Yaskawa INFORM job: KRIS8-PODLUZNCA_NEW.JBI

/JOB
//NAME KRIS8-PODLUZNCA_NEW
//POS
///NPOS 200,200,200,13,0,0
///TOOL 0
///POSTYPE PULSE
///PULSE
C00000=1998,-113620,-91819,0,89171,2
C00001=1998,-113620,-91819,0,89171,2
C00002=1998,-113620,-91819,0,89171,2
C00003=-50148,47658,9015,-3478,103612,-52965
C00004=-87671,10112,-26644,4452,101827,-68771
C00005=-89510,7784,-25446,4619,99998,-69437
C00006=-89510,7526,-24742,4610,99434,-69459
C00007=-89510,7784,-25446,4619,99998,-69437
C00008=-89141,5759,-27209,4581,100025,-69316
C00009=-89510,7784,-25446,4619,99998,-69437
C00010=-118549,-7920,-36001,7391,100506,-78970
C00011=-118558,-8065,-31852,7324,97901,-79128
C00012=-118558,-8215,-30981,7313,97294,-79164
C00013=-118558,-8065,-31852,7324,97901,-79128
C00014=-118526,-10509,-33773,7321,97825,-79123
C00015=-118558,-8065,-31852,7324,97901,-79128
C00016=-118558,-6729,-36855,7427,101637,-78904
C00017=-99982,-14384,-32914,3812,87667,-73559
C00018=-100648,-9156,-23354,4670,87204,-73724
C00019=-100648,-9135,-22594,4670,86748,-73740
C00020=-100648,-9156,-23354,4670,87204,-73724
C00021=-100304,-11982,-25556,4620,87088,-73613
C00022=-100648,-9156,-23354,4670,87204,-73724
C00023=-126523,-14506,-29918,8084,90525,-82231
C00024=-126543,-14617,-21806,8089,85527,-82559
C00025=-126543,-14515,-21015,8091,85096,-82587
C00026=-126543,-14617,-21806,8089,85527,-82559
C00027=-126622,-16805,-23452,8098,85423,-82593
C00028=-126543,-14617,-21806,8089,85527,-82559
C00029=-126543,-15095,-29845,8084,90184,-82258
C00030=-141008,-142584,-88347,10734,62671,-89412
C00031=-2633,-142584,-88347,10734,62671,-89412
C00032=-538,152103,58256,11565,122730,-83592
C00033=-538,152103,58256,11565,122730,-83592
C00034=-538,163731,66428,11721,123660,-83483
C00035=-24110,80646,-6840,3666,118579,-81953
C00036=-70155,49076,-66751,3666,118579,-81953
C00037=-75302,69312,-21887,-16743,132273,-74648
C00038=-73641,66162,-19190,-16029,129345,-73576
C00039=-73641,65328,-19214,-15924,128944,-73508
C00040=-74175,68002,-17054,-15046,130211,-73509
C00041=-73715,66523,-18896,-15177,130633,-73426
C00042=-74175,68002,-17054,-15046,130211,-73509
C00043=-74175,75772,-16365,-16008,133654,-74118
C00044=-92792,60028,-40452,-15957,137944,-80854
C00045=-92792,54549,-41170,-15193,135653,-80408
C00046=-92792,53504,-41275,-15052,135198,-80323
C00047=-92792,54549,-41170,-15193,135653,-80408
C00048=-92488,53114,-42914,-15337,136011,-80380
C00049=-92792,54549,-41170,-15193,135653,-80408
C00050=-92792,27665,-39260,-12049,121058,-78294
C00051=-132608,13603,-46395,-6888,114515,-90217
C00052=-132421,12280,-41624,-6966,112053,-90060
C00053=-132421,11796,-41286,-6941,111598,-90034
C00054=-132421,12280,-41624,-6966,112053,-90060
C00055=-132588,9844,-43810,-6954,112133,-90118
C00056=-132421,12280,-41624,-6966,112053,-90060
C00057=-132421,20626,-45689,-7423,118793,-90495
C00058=-93642,14896,-51087,-11726,122768,-78621
C00059=-121167,7250,-60994,-9109,122189,-87287
C00060=-121133,19973,-49305,-9042,121542,-87220
C00061=-121132,14285,-46771,-8609,117111,-86854
C00062=-121132,13713,-46508,-8571,116661,-86819
C00063=-121132,14285,-46771,-8609,117111,-86854
C00064=-121135,12460,-48440,-8614,117198,-86860
C00065=-121132,14285,-46771,-8609,117111,-86854
C00066=-121132,17545,-48059,-8835,119552,-87051
C00067=-132875,22669,-43773,5943,121981,-86806
C00068=-135068,19005,-43202,8732,120135,-86865
C00069=-125533,16786,-42812,7853,119266,-83887
C00070=-129035,15453,-41030,19832,117551,-82149
C00071=-130355,18004,-41916,20330,119568,-82220
C00072=-130907,11274,-51649,20974,122055,-81903
C00073=-97666,14619,-44772,-31513,122541,-85138
C00074=-89089,20309,-29812,-48880,120265,-85971
C00075=-90138,26219,-24118,-48560,119457,-86029
C00076=-94354,21466,-28820,-38570,118301,-84723
C00077=-94339,20725,-28307,-38311,117755,-84491
C00078=-97943,20254,-33169,-26633,118711,-83166
C00079=-102801,18851,-37203,-11200,118340,-81013
C00080=-105344,17460,-38317,-1076,116820,-79338
C00081=-107629,15720,-38660,7756,114602,-78025
C00082=-107337,17368,-35211,13069,113626,-76697
C00083=-107325,21456,-38051,13546,117374,-76240
C00084=-114827,9197,-39078,13016,110805,-79564
C00085=-114816,5999,-36185,12673,107231,-79960
C00086=-89500,15411,-20924,8846,98241,-72558
C00087=-89521,17497,-24405,8955,101422,-72333
C00088=-120014,-138037,-117853,25062,55116,-87984
C00089=-139340,-34559,-66869,29462,80713,-89295
C00090=-144770,-30804,-73292,39943,77473,-90359
C00091=-143362,-21275,-66712,39157,77581,-89780
C00092=-144483,-24614,-74965,39351,80645,-89055
C00093=-151238,-55243,-102038,42556,83965,-90229
C00094=10330,-8063,-71326,-50992,95178,-51096
C00095=10330,-154777,-122755,75707,95178,-51096
C00096=10330,-154777,-122755,75707,95178,-51096
C00097=-84612,8206,-36800,5840,103129,-68484
C00098=-86865,7918,-29603,3944,101662,-68585
C00099=-87828,11476,-22006,5366,101518,-68689
C00100=-118917,-5972,-29345,7466,99945,-79124
C00101=-118924,-4449,-32352,7580,103027,-78936
C00102=-137167,-2659,-36348,8728,105802,-84843
C00103=-109963,-5720,-34048,6846,100758,-76100
C00104=-138502,-3992,-26225,8429,99500,-85759
C00105=-138502,843,-39441,8925,110003,-85001
C00106=-88254,-47088,-61974,-10192,62970,-70123
C00107=-81608,-29587,-43634,-21841,66061,-69208
C00108=-83532,-22198,-38463,-20877,66146,-69964
C00109=-81853,-28331,-46732,-21354,68381,-69747
C00110=-4657,-138190,-117116,-41247,88176,-44256
C00111=1998,-113620,-91819,0,89171,2
C00112=-50148,47658,9015,-3478,103612,-52965
C00113=-122206,-8197,-37642,7697,101693,-80109
C00114=-122172,-5530,-28898,7592,99531,-80240
C00115=-122172,-5644,-28166,7579,99029,-80270
C00116=-122172,-5530,-28898,7592,99531,-80240
C00117=-122187,-7349,-30356,7592,99495,-80247
C00118=-122172,-5530,-28898,7592,99531,-80240
C00119=-152388,7436,-14473,8976,99151,-90470
C00120=-152540,6439,-11770,9191,96395,-90696
C00121=-152540,6437,-10968,9184,95908,-90732
C00122=-152540,6439,-11770,9191,96395,-90696
C00123=-152857,4706,-13266,9200,96461,-90799
C00124=-152540,6439,-11770,9191,96395,-90696
C00125=-152540,6878,-17750,9308,100253,-90406
C00126=-127365,-8235,-30314,7954,97587,-82094
C00127=-127365,-8135,-15746,8070,86282,-82798
C00128=-127365,-8012,-14852,8071,85798,-82829
C00129=-127365,-8135,-15746,8070,86282,-82798
C00130=-127450,-10284,-17434,8077,86227,-82833
C00131=-127365,-8135,-15746,8070,86282,-82798
C00132=-126523,-14506,-29918,8084,90525,-82231
C00133=-123077,-8463,-14980,-23626,83972,-82532
C00134=-125016,-5406,-1705,-27943,77200,-81831
C00135=-125016,-5123,-715,-27989,76788,-81729
C00136=-125016,-5449,-1860,-27937,77265,-81847
C00137=-125063,-7239,-3294,-27936,77216,-81852
C00138=-125016,-5449,-1860,-27937,77265,-81847
C00139=-125016,-6433,-5581,-27781,78853,-82232
C00140=-141008,-142584,-88347,10734,62671,-89412
C00141=-2633,-142584,-88347,10734,62671,-89412
C00142=-538,152103,58256,11565,122730,-83592
C00143=-538,152103,58256,11565,122730,-83592
C00144=-538,163731,66428,11721,123660,-83483
C00145=-24110,80646,-6840,3666,118579,-81953
C00146=-70155,49076,-66751,3666,118579,-81953
C00147=-75302,69312,-21887,-16743,132273,-74648
C00148=-71157,73317,-9100,-15659,127243,-72407
C00149=-71157,72393,-9111,-15553,126791,-72333
C00150=-71157,73317,-9100,-15659,127243,-72407
C00151=-70763,72072,-10673,-15771,127615,-72338
C00152=-71157,73317,-9100,-15659,127243,-72407
C00153=-71157,75512,-9016,-15913,128280,-72581
C00154=-70753,69276,-8084,9618,109691,-64304
C00155=-70054,68719,-6250,9333,108233,-64227
C00156=-70054,67798,-6136,9301,107694,-64269
C00157=-70054,68719,-6250,9333,108233,-64227
C00158=-69682,67506,-7733,9249,108486,-64104
C00159=-70054,68719,-6250,9333,108233,-64227
C00160=-71410,68261,-9608,9830,110161,-64447
C00161=-100211,16967,-41384,-5250,115146,-78637
C00162=-100101,13848,-40894,-5174,113254,-78516
C00163=-100101,13093,-40376,-5142,112548,-78482
C00164=-100101,13848,-40894,-5174,113254,-78516
C00165=-99916,12326,-42277,-5198,113335,-78462
C00166=-100101,13848,-40894,-5174,113254,-78516
C00167=-128373,12968,-45365,-6146,114904,-88569
C00168=-128373,11236,-44374,-6065,113413,-88488
C00169=-128373,10392,-43832,-6025,112650,-88447
C00170=-128373,11236,-44374,-6065,113413,-88488
C00171=-128461,9274,-46126,-6059,113476,-88521
C00172=-128373,11236,-44374,-6065,113413,-88488
C00173=-126467,9541,-45537,-4537,113892,-87464
C00174=-90696,17389,-28668,-7563,109954,-75731
C00175=-90696,19081,-30431,-7676,111892,-75859
C00176=-95392,14915,-34303,-7326,111749,-77384
C00177=-94182,13407,-27747,-8042,105770,-76801
C00178=-94182,12413,-26084,-7974,104249,-76699
C00179=-87479,17429,-16267,6238,94957,-72183
C00180=-90143,10225,-11740,26784,78164,-72685
C00181=-93708,-8754,-29680,24752,70317,-76342
C00182=-120014,-138037,-117853,25062,55116,-87984
C00183=10330,-8063,-71326,-50992,95178,-51096
C00184=10330,-154777,-122755,75707,95178,-51096
C00185=10330,-154777,-122755,75707,95178,-51096
C00186=-115154,-11106,-52771,10493,105816,-77983
C00187=-114081,-13344,-38355,9938,95819,-78468
C00188=-107530,-11938,-34647,9052,93539,-76468
C00189=-146196,-5358,-20976,12882,93830,-89505
C00190=-146196,-5254,-24370,12940,95920,-89287
C00191=-128813,-13564,-32541,11522,94088,-83555
C00192=-121674,-10043,-17729,10735,85943,-81851
C00193=-132101,-7653,-13572,11769,86087,-85426
C00194=-123125,-7882,-8368,-19622,80618,-82966
C00195=-119420,-3587,6095,-39306,76343,-80043
C00196=-113107,-5257,-1068,-39217,81983,-79383
C00197=-103899,-33329,-43273,-25917,82676,-77420
C00198=-4657,-138190,-117116,-41247,88176,-44256
C00199=1998,-113620,-91819,0,89171,2
BC00000=87190,689489,1075225
BC00001=87190,689489,1075225
BC00002=87190,689489,1075225
BC00003=205563,689489,1075225
BC00004=321532,689489,1014461
BC00005=321532,689488,1014457
BC00006=321532,689488,1014457
BC00007=321532,689488,1014457
BC00008=321532,689488,1014457
BC00009=321532,689488,1014457
BC00010=321532,689488,1014457
BC00011=321532,689488,1014457
BC00012=321532,689488,1014457
BC00013=321532,689488,1014457
BC00014=321532,689488,1014457
BC00015=321532,689488,1014457
BC00016=321532,689488,1014457
BC00017=179819,689488,1014457
BC00018=179819,689488,1014457
BC00019=179819,689488,1014457
BC00020=179819,689488,1014457
BC00021=179819,689488,1014457
BC00022=179819,689488,1014457
BC00023=179819,689488,1014457
BC00024=179819,689488,1014457
BC00025=179819,689488,1014457
BC00026=179819,689488,1014457
BC00027=179819,689488,1014457
BC00028=179819,689488,1014457
BC00029=179819,689488,1014457
BC00030=179819,689488,1014456
BC00031=179819,689488,1014456
BC00032=179819,689488,1014456
BC00033=179819,689488,1014456
BC00034=117363,689487,547728
BC00035=117363,689487,547728
BC00036=117363,689487,547728
BC00037=137555,679820,547728
BC00038=137555,679820,547728
BC00039=137555,679820,547728
BC00040=137555,679820,547728
BC00041=137555,679820,547728
BC00042=137555,679820,547728
BC00043=137555,679820,547728
BC00044=137555,679820,547728
BC00045=137555,679820,547728
BC00046=137555,679820,547728
BC00047=137555,679820,547728
BC00048=137555,679820,547728
BC00049=137555,679820,547728
BC00050=137555,679820,764194
BC00051=137555,679820,847065
BC00052=137555,679820,847065
BC00053=137555,679820,847065
BC00054=137555,679820,847065
BC00055=137555,679820,847065
BC00056=137555,679820,847065
BC00057=137555,679820,847065
BC00058=39902,679820,847065
BC00059=39902,679820,847065
BC00060=39902,679820,847065
BC00061=39902,679820,847065
BC00062=39902,679820,847065
BC00063=39902,679820,847065
BC00064=39902,679820,847065
BC00065=39902,679820,847065
BC00066=39902,679820,847065
BC00067=39902,679820,847065
BC00068=39902,679820,847065
BC00069=39902,679820,847065
BC00070=39902,679821,847064
BC00071=39902,679821,847064
BC00072=39902,679821,847064
BC00073=39902,679821,847064
BC00074=39902,679821,847064
BC00075=39902,679821,847064
BC00076=39902,679821,847064
BC00077=39902,679821,847064
BC00078=39902,679821,847064
BC00079=39902,679821,847064
BC00080=39902,679821,847064
BC00081=39902,679821,847064
BC00082=39902,679821,847064
BC00083=39902,679821,847064
BC00084=153593,679821,847061
BC00085=153593,679821,847061
BC00086=153593,679821,847061
BC00087=153593,679821,847061
BC00088=153593,679821,847061
BC00089=153593,679821,847061
BC00090=153593,679821,675096
BC00091=153593,679821,675096
BC00092=153593,679821,675096
BC00093=153593,679821,675096
BC00094=153593,679821,675096
BC00095=21039,679821,892901
BC00096=21039,679821,892901
BC00097=305234,688965,1007868
BC00098=321532,689489,1014461
BC00099=321532,689489,1014461
BC00100=321532,689489,1014461
BC00101=321532,689489,1014461
BC00102=271871,689488,929443
BC00103=205923,689488,929443
BC00104=205923,689488,929443
BC00105=205923,689488,929443
BC00106=205923,689488,929443
BC00107=205923,689488,929443
BC00108=205923,689488,929443
BC00109=205923,689488,929443
BC00110=205923,689488,929443
BC00111=87190,689489,1075225
BC00112=205563,689489,1075225
BC00113=321532,689489,1014458
BC00114=321532,689489,1014458
BC00115=321532,689489,1014458
BC00116=321532,689489,1014458
BC00117=321532,689489,1014458
BC00118=321532,689489,1014458
BC00119=321531,689488,1014455
BC00120=321531,689488,1014455
BC00121=321531,689488,1014455
BC00122=321531,689488,1014455
BC00123=321531,689488,1014455
BC00124=321531,689488,1014455
BC00125=321531,689488,1014455
BC00126=168038,689488,1014455
BC00127=168038,689488,1014455
BC00128=168038,689488,1014455
BC00129=168038,689488,1014455
BC00130=168038,689488,1014455
BC00131=168038,689488,1014455
BC00132=179819,689488,1014457
BC00133=168038,689488,1014455
BC00134=168038,689488,1014455
BC00135=168038,689488,1014455
BC00136=168038,689488,1014455
BC00137=168038,689488,1014455
BC00138=168038,689488,1014455
BC00139=168038,689488,1014455
BC00140=179819,689488,1014456
BC00141=179819,689488,1014456
BC00142=179819,689488,1014456
BC00143=179819,689488,1014456
BC00144=117363,689487,547728
BC00145=117363,689487,547728
BC00146=117363,689487,547728
BC00147=137555,679820,547728
BC00148=137555,679820,547728
BC00149=137555,679820,547728
BC00150=137555,679820,547728
BC00151=137555,679820,547728
BC00152=137555,679820,547728
BC00153=137555,679820,547728
BC00154=137555,679820,547728
BC00155=137555,679820,547728
BC00156=137555,679820,547728
BC00157=137555,679820,547728
BC00158=137555,679820,547728
BC00159=137555,679820,547728
BC00160=137555,679820,547728
BC00161=137555,679820,790702
BC00162=137555,679820,790702
BC00163=137555,679820,790702
BC00164=137555,679820,790702
BC00165=137555,679820,790702
BC00166=137555,679820,790702
BC00167=137555,679820,832612
BC00168=137555,679820,832612
BC00169=137555,679820,832612
BC00170=137555,679820,832612
BC00171=137555,679820,832612
BC00172=137555,679820,832612
BC00173=122098,679820,834897
BC00174=122098,679820,834897
BC00175=122098,679820,834897
BC00176=205006,679820,834897
BC00177=205006,679820,834897
BC00178=205006,679820,834897
BC00179=205006,679820,834897
BC00180=205006,679820,834897
BC00181=205006,679820,834897
BC00182=153593,679821,847061
BC00183=153593,679821,675096
BC00184=21039,679821,892901
BC00185=21039,679821,892901
BC00186=305234,688965,1007868
BC00187=305234,688965,1007868
BC00188=289400,688965,1007868
BC00189=289400,688965,1007868
BC00190=289400,688965,1007868
BC00191=153159,688965,1007868
BC00192=153159,688965,1007868
BC00193=153159,688965,1007868
BC00194=153159,688965,1007868
BC00195=153159,688965,1007868
BC00196=153159,688965,1007868
BC00197=171750,689149,980236
BC00198=205923,689488,929443
BC00199=87190,689489,1075225
EC00000=1,0
EC00001=-1596314,0
EC00002=-1596314,0
EC00003=-1596314,0
EC00004=-1596314,0
EC00005=-1596314,0
EC00006=-1596314,0
EC00007=-1596314,0
EC00008=-1596314,0
EC00009=-1596314,0
EC00010=-1596314,0
EC00011=-1596314,0
EC00012=-1596314,0
EC00013=-1596314,0
EC00014=-1596314,0
EC00015=-1596314,0
EC00016=-1596314,0
EC00017=-1596314,0
EC00018=-1596314,0
EC00019=-1596314,0
EC00020=-1596314,0
EC00021=-1596314,0
EC00022=-1596314,0
EC00023=-1596314,0
EC00024=-1596314,0
EC00025=-1596314,0
EC00026=-1596314,0
EC00027=-1596314,0
EC00028=-1596314,0
EC00029=-1596314,0
EC00030=-1596314,1
EC00031=-1596314,1
EC00032=-1596314,1
EC00033=-1596314,1112952
EC00034=-1596313,1112949
EC00035=-1596313,1112949
EC00036=-1596313,1112949
EC00037=-1596313,1112949
EC00038=-1596313,1112949
EC00039=-1596313,1112949
EC00040=-1596313,1112949
EC00041=-1596313,1112949
EC00042=-1596313,1112949
EC00043=-1596313,1112949
EC00044=-1596313,1112949
EC00045=-1596313,1112949
EC00046=-1596313,1112949
EC00047=-1596313,1112949
EC00048=-1596313,1112949
EC00049=-1596313,1112949
EC00050=-1596313,1112949
EC00051=-1596313,1112949
EC00052=-1596313,1112949
EC00053=-1596313,1112949
EC00054=-1596313,1112949
EC00055=-1596313,1112949
EC00056=-1596313,1112949
EC00057=-1596313,1112949
EC00058=-1596313,1112949
EC00059=-1596313,1112949
EC00060=-1596313,1112949
EC00061=-1596313,1112949
EC00062=-1596313,1112949
EC00063=-1596313,1112949
EC00064=-1596313,1112949
EC00065=-1596313,1112949
EC00066=-1596313,1112949
EC00067=-1596313,1112949
EC00068=-1596313,1112949
EC00069=-1596313,1112949
EC00070=-1596313,1112949
EC00071=-1596313,1112949
EC00072=-1596313,1112949
EC00073=-1596313,1112949
EC00074=-1596313,1112949
EC00075=-1596313,1112949
EC00076=-1596313,1112949
EC00077=-1596313,1112949
EC00078=-1596313,1112949
EC00079=-1596313,1112949
EC00080=-1596313,1112949
EC00081=-1596313,1112949
EC00082=-1596313,1112949
EC00083=-1596313,1112949
EC00084=-1596313,1112949
EC00085=-1596313,1112949
EC00086=-1596313,1112949
EC00087=-1596313,1112949
EC00088=-1596313,1112949
EC00089=-1596313,1112949
EC00090=-1596313,1112949
EC00091=-1596313,1112949
EC00092=-1596313,1112949
EC00093=-1596313,1112949
EC00094=-1596313,1112949
EC00095=-1596313,1112949
EC00096=-1596313,0
EC00097=-1596314,0
EC00098=-1596314,0
EC00099=-1596314,0
EC00100=-1596314,0
EC00101=-1596314,0
EC00102=-1596314,0
EC00103=-1596314,0
EC00104=-1596314,0
EC00105=-1596314,0
EC00106=-1596314,0
EC00107=-1596314,0
EC00108=-1596314,0
EC00109=-1596314,0
EC00110=-1596314,0
EC00111=-1596314,0
EC00112=-1596314,0
EC00113=-1596314,0
EC00114=-1596314,0
EC00115=-1596314,0
EC00116=-1596314,0
EC00117=-1596314,0
EC00118=-1596314,0
EC00119=-1596315,0
EC00120=-1596315,0
EC00121=-1596315,0
EC00122=-1596315,0
EC00123=-1596315,0
EC00124=-1596315,0
EC00125=-1596315,0
EC00126=-1596315,0
EC00127=-1596315,0
EC00128=-1596315,0
EC00129=-1596315,0
EC00130=-1596315,0
EC00131=-1596315,0
EC00132=-1596314,0
EC00133=-1596315,0
EC00134=-1596315,0
EC00135=-1596315,0
EC00136=-1596315,0
EC00137=-1596315,0
EC00138=-1596315,0
EC00139=-1596315,0
EC00140=-1596314,1
EC00141=-1596314,1
EC00142=-1596314,1
EC00143=-1596314,1112952
EC00144=-1596313,1112949
EC00145=-1596313,1112949
EC00146=-1596313,1112949
EC00147=-1596313,1112949
EC00148=-1596313,1112949
EC00149=-1596313,1112949
EC00150=-1596313,1112949
EC00151=-1596313,1112949
EC00152=-1596313,1112949
EC00153=-1596313,1112949
EC00154=-1596313,1112949
EC00155=-1596313,1112949
EC00156=-1596313,1112949
EC00157=-1596313,1112949
EC00158=-1596313,1112949
EC00159=-1596313,1112949
EC00160=-1596313,1112949
EC00161=-1596313,1112949
EC00162=-1596313,1112949
EC00163=-1596313,1112949
EC00164=-1596313,1112949
EC00165=-1596313,1112949
EC00166=-1596313,1112949
EC00167=-1596313,1112949
EC00168=-1596313,1112949
EC00169=-1596313,1112949
EC00170=-1596313,1112949
EC00171=-1596313,1112949
EC00172=-1596313,1112949
EC00173=-1596313,1112949
EC00174=-1596313,1112949
EC00175=-1596313,1112949
EC00176=-1596313,1112949
EC00177=-1596313,1112949
EC00178=-1596313,1112949
EC00179=-1596313,1112949
EC00180=-1596313,1112949
EC00181=-1596313,1112949
EC00182=-1596313,1112949
EC00183=-1596313,1112949
EC00184=-1596313,1112949
EC00185=-1596313,0
EC00186=-1596314,0
EC00187=-1596314,0
EC00188=-1596314,0
EC00189=-1596314,0
EC00190=-1596314,0
EC00191=-1596314,0
EC00192=-1596314,0
EC00193=-1596314,0
EC00194=-1596314,0
EC00195=-1596314,0
EC00196=-1596314,0
EC00197=-1596314,0
EC00198=-1596314,0
EC00199=1,0
///POSTYPE BASE
///RECTAN
///RCONF 0,0,0,0,0,0,0,0,0,0,0,0,0,0,0,0,0,0,0,0,0,0,0,0
P00006=0.145,-0.552,1.326,0.0000,0.0000,0.0000
P00021=-0.339,1.359,3.368,0.0000,0.0000,0.0000
P00022=-0.114,-0.780,3.887,0.0000,0.0000,0.0000
P00023=0.143,-0.036,0.682,0.0000,0.0000,0.0000
P00024=0.145,-0.552,1.326,0.0000,0.0000,0.0000
P00025=2.242,-0.049,-1.961,0.0000,0.0000,0.0000
P00026=0.572,-0.002,0.234,0.0000,0.0000,0.0000
P00027=-0.746,0.015,-9.096,0.0000,0.0000,0.0000
P00028=-2.237,-0.018,-7.702,0.0000,0.0000,0.0000
P00031=1.853,-0.001,-1.549,0.0000,0.0000,0.0000
P00032=1.957,0.503,-7.217,0.0000,0.0000,0.0000
///RCONF 0,0,0,0,1,0,0,0,0,0,0,0,0,0,0,0,0,0,0,0,0,0,0,0
P00033=-0.123,0.612,-5.012,0.0000,0.0000,0.0000
///RCONF 0,0,0,0,0,0,0,0,0,0,0,0,0,0,0,0,0,0,0,0,0,0,0,0
P00034=-0.304,0.773,-2.693,0.0000,0.0000,0.0000
//INST
///DATE 2024/02/26 20:33
///ATTR SC,RW
///GROUP1 RB1,BS1
///GROUP2 ST1
NOP
MOVJ C00000 BC00000 VJ=100.00  +MOVJ EC00000 VJ=100.00
MOVJ C00001 BC00001 VJ=100.00  +MOVJ EC00001 VJ=100.00
CALL JOB:CLEAN-R1_KM_NEW
MOVJ C00002 BC00002 VJ=100.00  +MOVJ EC00002 VJ=100.00
MOVJ C00003 BC00003 VJ=100.00  +MOVJ EC00003 VJ=15.00
SMOVL C00004 BC00004 V=100.0  +MOVJ EC00004
SMOVL C00005 BC00005 V=100.0  +MOVJ EC00005
SREFP 3 C00006 BC00006  +REFP EC00006
CALL JOB:SEARCH-R1-S1
SET P021 P006
SSFTON P021
SMOVL C00007 BC00007 V=100.0  +MOVJ EC00007
SREFP 3 C00008 BC00008  +REFP EC00008
CALL JOB:SEARCH-R1-S1
SET P021 P006
SSFTON P021
SMOVL C00009 BC00009 V=133.3  +MOVJ EC00009
SSFTOF
SMOVL C00010 BC00010 V=266.7  +MOVJ EC00010
SMOVL C00011 BC00011 V=100.0  +MOVJ EC00011
SREFP 3 C00012 BC00012  +REFP EC00012
CALL JOB:SEARCH-R1-S1
SET P022 P006
SSFTON P022
SMOVL C00013 BC00013 V=100.0  +MOVJ EC00013
SREFP 3 C00014 BC00014  +REFP EC00014
CALL JOB:SEARCH-R1-S1
SET P022 P006
SSFTON P022
SMOVL C00015 BC00015 V=133.3  +MOVJ EC00015
SSFTOF
SMOVL C00016 BC00016 V=266.7  +MOVJ EC00016
SMOVL C00017 BC00017 V=266.7  +MOVJ EC00017
SMOVL C00018 BC00018 V=100.0  +MOVJ EC00018
SREFP 3 C00019 BC00019  +REFP EC00019
CALL JOB:SEARCH-R1-S1
SET P023 P006
SSFTON P023
SMOVL C00020 BC00020 V=100.0  +MOVJ EC00020
SREFP 3 C00021 BC00021  +REFP EC00021
CALL JOB:SEARCH-R1-S1
SET P023 P006
SSFTON P023
SMOVL C00022 BC00022 V=133.3  +MOVJ EC00022
SSFTOF
SMOVL C00023 BC00023 V=266.7  +MOVJ EC00023
SMOVL C00024 BC00024 V=100.0  +MOVJ EC00024
SREFP 3 C00025 BC00025  +REFP EC00025
CALL JOB:SEARCH-R1-S1
SET P024 P006
SSFTON P024
SMOVL C00026 BC00026 V=100.0  +MOVJ EC00026
SREFP 3 C00027 BC00027  +REFP EC00027
CALL JOB:SEARCH-R1-S1
SET P024 P006
SSFTON P024
SMOVL C00028 BC00028 V=133.3  +MOVJ EC00028
SSFTOF
SMOVL C00029 BC00029 V=266.7  +MOVJ EC00029
SMOVL C00030 BC00030 V=666.7  +MOVJ EC00030
MOVJ C00031 BC00031 VJ=100.00  +MOVJ EC00031 VJ=100.00
MOVJ C00032 BC00032 VJ=100.00  +MOVJ EC00032 VJ=100.00
'OBROT
MOVJ C00033 BC00033 VJ=100.00  +MOVJ EC00033 VJ=100.00
MOVJ C00034 BC00034 VJ=100.00  +MOVJ EC00034 VJ=100.00
MOVJ C00035 BC00035 VJ=100.00  +MOVJ EC00035 VJ=100.00
MOVJ C00036 BC00036 VJ=100.00  +MOVJ EC00036 VJ=100.00
MOVJ C00037 BC00037 VJ=100.00  +MOVJ EC00037 VJ=100.00
SMOVL C00038 BC00038 V=100.0  +MOVJ EC00038
SREFP 3 C00039 BC00039  +REFP EC00039
CALL JOB:SEARCH-R1-S1
SET P025 P006
SSFTON P025
SMOVL C00040 BC00040 V=100.0  +MOVJ EC00040
SREFP 3 C00041 BC00041  +REFP EC00041
CALL JOB:SEARCH-R1-S1
SET P025 P006
SSFTON P025
SMOVL C00042 BC00042 V=133.3  +MOVJ EC00042
SSFTOF
SMOVL C00043 BC00043 V=266.7  +MOVJ EC00043
SMOVL C00044 BC00044 V=266.7  +MOVJ EC00044
SMOVL C00045 BC00045 V=100.0  +MOVJ EC00045
SREFP 3 C00046 BC00046  +REFP EC00046
CALL JOB:SEARCH-R1-S1
SET P026 P006
SSFTON P026
SMOVL C00047 BC00047 V=100.0  +MOVJ EC00047
SREFP 3 C00048 BC00048  +REFP EC00048
CALL JOB:SEARCH-R1-S1
SET P026 P006
SSFTON P026
SMOVL C00049 BC00049 V=133.3  +MOVJ EC00049
SSFTOF
SMOVL C00050 BC00050 V=266.7  +MOVJ EC00050
SMOVL C00051 BC00051 V=266.7  +MOVJ EC00051
SMOVL C00052 BC00052 V=100.0  +MOVJ EC00052
SREFP 3 C00053 BC00053  +REFP EC00053
CALL JOB:SEARCH-R1-S1
SET P027 P006
SSFTON P027
SMOVL C00054 BC00054 V=100.0  +MOVJ EC00054
SREFP 3 C00055 BC00055  +REFP EC00055
CALL JOB:SEARCH-R1-S1
SET P027 P006
SSFTON P027
SMOVL C00056 BC00056 V=133.3  +MOVJ EC00056
SSFTOF
SMOVL C00057 BC00057 V=266.7  +MOVJ EC00057
SMOVL C00058 BC00058 V=266.7  +MOVJ EC00058
SMOVL C00059 BC00059 V=266.7  +MOVJ EC00059
SMOVL C00060 BC00060 V=266.7  +MOVJ EC00060
SMOVL C00061 BC00061 V=100.0  +MOVJ EC00061
SREFP 3 C00062 BC00062  +REFP EC00062
CALL JOB:SEARCH-R1-S1
SET P028 P006
SSFTON P028
SMOVL C00063 BC00063 V=100.0  +MOVJ EC00063
SREFP 3 C00064 BC00064  +REFP EC00064
CALL JOB:SEARCH-R1-S1
SET P028 P006
SSFTON P028
SMOVL C00065 BC00065 V=133.3  +MOVJ EC00065
SSFTOF
SMOVL C00066 BC00066 V=266.7  +MOVJ EC00066
SMOVL C00067 BC00067 V=266.7  +MOVJ EC00067
SSFTON P028
MACRO1 MJ#(0) ARGF6
SMOVL C00068 BC00068 V=100.0  +MOVJ EC00068
ARCON
SWVON WEV#(50)
SMOVL C00069 BC00069 V=7.5  +MOVJ EC00069
SMOVL C00070 BC00070 V=7.5  +MOVJ EC00070
ARCOF
SWVOF
SMOVL C00071 BC00071 V=100.0  +MOVJ EC00071
SSFTOF
SMOVL C00072 BC00072 V=100.0  +MOVJ EC00072
SMOVL C00073 BC00073 V=100.0  +MOVJ EC00073
SMOVL C00074 BC00074 V=100.0  +MOVJ EC00074
SMOVL C00075 BC00075 V=100.0  +MOVJ EC00075
SMOVL C00076 BC00076 V=100.0  +MOVJ EC00076
SSFTON P027
SMOVL C00077 BC00077 V=100.0  +MOVJ EC00077
ARCON
SMOVL C00078 BC00078 V=6.7  +MOVJ EC00078
SMOVL C00079 BC00079 V=6.7  +MOVJ EC00079
SMOVL C00080 BC00080 V=6.7  +MOVJ EC00080
SMOVL C00081 BC00081 V=6.7  +MOVJ EC00081
SMOVL C00082 BC00082 V=6.7  +MOVJ EC00082
ARCOF
SMOVL C00083 BC00083 V=133.3  +MOVJ EC00083
SSFTOF
SMOVL C00084 BC00084 V=266.7  +MOVJ EC00084
SSFTON P026
SMOVL C00085 BC00085 V=100.0  +MOVJ EC00085
ARCON
SWVON WEV#(50)
SSFTON P025
SMOVL C00086 BC00086 V=7.0  +MOVJ EC00086
ARCOF
SMOVL C00087 BC00087 V=133.3  +MOVJ EC00087
SSFTOF
SMOVL C00088 BC00088 V=666.7  +MOVJ EC00088
SMOVL C00089 BC00089 V=666.7  +MOVJ EC00089
MACRO1 MJ#(0) ARGF14
SMOVL C00090 BC00090 V=100.0  +MOVJ EC00090
ARCON
SWVON WEV#(40)
SMOVL C00091 BC00091 V=7.5  +MOVJ EC00091
ARCOF
SWVOF
SMOVL C00092 BC00092 V=133.3  +MOVJ EC00092
SMOVL C00093 BC00093 V=666.7  +MOVJ EC00093
MOVJ C00094 BC00094 VJ=100.00  +MOVJ EC00094 VJ=100.00
MOVJ C00095 BC00095 VJ=100.00  +MOVJ EC00095 VJ=100.00
MOVJ C00096 BC00096 VJ=100.00  +MOVJ EC00096 VJ=100.00
MOVJ C00097 BC00097 VJ=100.00  +MOVJ EC00097 VJ=100.00
SMOVL C00098 BC00098 V=100.0  +MOVJ EC00098
MACRO1 MJ#(0) ARGF14
SSFTON P021
SMOVL C00099 BC00099 V=100.0  +MOVJ EC00099
ARCON
SWVON WEV#(50)
SSFTON P022
SMOVL C00100 BC00100 V=10.0  +MOVJ EC00100
ARCOF
SWVOF
SMOVL C00101 BC00101 V=266.7  +MOVJ EC00101
SSFTOF
SMOVL C00102 BC00102 V=266.7  +MOVJ EC00102
SSFTON P023
SMOVL C00103 BC00103 V=100.0  +MOVJ EC00103
ARCON
SWVON WEV#(50)
SSFTON P024
SMOVL C00104 BC00104 V=9.2  +MOVJ EC00104
ARCOF
SWVOF
SMOVL C00105 BC00105 V=266.7  +MOVJ EC00105
SSFTOF
SMOVL C00106 BC00106 V=266.7  +MOVJ EC00106
SMOVL C00107 BC00107 V=100.0  +MOVJ EC00107
ARCON
SWVON WEV#(40)
SMOVL C00108 BC00108 V=7.5  +MOVJ EC00108
ARCOF
SWVOF
SMOVL C00109 BC00109 V=266.7  +MOVJ EC00109
SMOVL C00110 BC00110 V=266.7  +MOVJ EC00110
CALL JOB:CLEAN-R1_KM_NEW
'COMMENT
'COMMENT
MOVJ C00111 BC00111 VJ=100.00  +MOVJ EC00111 VJ=100.00
MOVJ C00112 BC00112 VJ=100.00  +MOVJ EC00112 VJ=15.00
SMOVL C00113 BC00113 V=100.0  +MOVJ EC00113
SMOVL C00114 BC00114 V=100.0  +MOVJ EC00114
SREFP 3 C00115 BC00115  +REFP EC00115
CALL JOB:SEARCH-R1-S1
SET P031 P006
SSFTON P031
SMOVL C00116 BC00116 V=100.0  +MOVJ EC00116
SREFP 3 C00117 BC00117  +REFP EC00117
CALL JOB:SEARCH-R1-S1
SET P031 P006
SSFTON P031
SMOVL C00118 BC00118 V=133.3  +MOVJ EC00118
SSFTOF
SMOVL C00119 BC00119 V=266.7  +MOVJ EC00119
SMOVL C00120 BC00120 V=100.0  +MOVJ EC00120
SREFP 3 C00121 BC00121  +REFP EC00121
CALL JOB:SEARCH-R1-S1
SET P032 P006
SSFTON P032
SMOVL C00122 BC00122 V=100.0  +MOVJ EC00122
SREFP 3 C00123 BC00123  +REFP EC00123
CALL JOB:SEARCH-R1-S1
SET P032 P006
SSFTON P032
SMOVL C00124 BC00124 V=133.3  +MOVJ EC00124
SSFTOF
SMOVL C00125 BC00125 V=266.7  +MOVJ EC00125
SMOVL C00126 BC00126 V=266.7  +MOVJ EC00126
SMOVL C00127 BC00127 V=100.0  +MOVJ EC00127
SREFP 3 C00128 BC00128  +REFP EC00128
CALL JOB:SEARCH-R1-S1
SET P033 P006
SSFTON P033
SMOVL C00129 BC00129 V=100.0  +MOVJ EC00129
SREFP 3 C00130 BC00130  +REFP EC00130
CALL JOB:SEARCH-R1-S1
SET P033 P006
SSFTON P033
SMOVL C00131 BC00131 V=133.3  +MOVJ EC00131
SSFTOF
SMOVL C00132 BC00132 V=266.7  +MOVJ EC00132
SMOVL C00133 BC00133 V=266.7  +MOVJ EC00133
SMOVL C00134 BC00134 V=100.0  +MOVJ EC00134
SREFP 3 C00135 BC00135  +REFP EC00135
CALL JOB:SEARCH-R1-S1
SET P034 P006
SSFTON P034
SMOVL C00136 BC00136 V=100.0  +MOVJ EC00136
SREFP 3 C00137 BC00137  +REFP EC00137
CALL JOB:SEARCH-R1-S1
SET P034 P006
SSFTON P034
SMOVL C00138 BC00138 V=133.3  +MOVJ EC00138
SSFTOF
SMOVL C00139 BC00139 V=266.7  +MOVJ EC00139
SMOVL C00140 BC00140 V=666.7  +MOVJ EC00140
MOVJ C00141 BC00141 VJ=100.00  +MOVJ EC00141 VJ=100.00
MOVJ C00142 BC00142 VJ=100.00  +MOVJ EC00142 VJ=100.00
'OBROT
MOVJ C00143 BC00143 VJ=100.00  +MOVJ EC00143 VJ=100.00
MOVJ C00144 BC00144 VJ=100.00  +MOVJ EC00144 VJ=100.00
MOVJ C00145 BC00145 VJ=100.00  +MOVJ EC00145 VJ=100.00
MOVJ C00146 BC00146 VJ=100.00  +MOVJ EC00146 VJ=100.00
MOVJ C00147 BC00147 VJ=100.00  +MOVJ EC00147 VJ=100.00
SMOVL C00148 BC00148 V=100.0  +MOVJ EC00148
SREFP 3 C00149 BC00149  +REFP EC00149
CALL JOB:SEARCH-R1-S1
SET P025 P006
SSFTON P025
SMOVL C00150 BC00150 V=100.0  +MOVJ EC00150
SREFP 3 C00151 BC00151  +REFP EC00151
CALL JOB:SEARCH-R1-S1
SET P025 P006
SSFTON P025
SMOVL C00152 BC00152 V=133.3  +MOVJ EC00152
SSFTOF
SMOVL C00153 BC00153 V=266.7  +MOVJ EC00153
SMOVL C00154 BC00154 V=266.7  +MOVJ EC00154
SMOVL C00155 BC00155 V=100.0  +MOVJ EC00155
SREFP 3 C00156 BC00156  +REFP EC00156
CALL JOB:SEARCH-R1-S1
SET P026 P006
SSFTON P026
SMOVL C00157 BC00157 V=100.0  +MOVJ EC00157
SREFP 3 C00158 BC00158  +REFP EC00158
CALL JOB:SEARCH-R1-S1
SET P026 P006
SSFTON P026
SMOVL C00159 BC00159 V=133.3  +MOVJ EC00159
SSFTOF
SMOVL C00160 BC00160 V=266.7  +MOVJ EC00160
SMOVL C00161 BC00161 V=266.7  +MOVJ EC00161
SMOVL C00162 BC00162 V=100.0  +MOVJ EC00162
SREFP 3 C00163 BC00163  +REFP EC00163
CALL JOB:SEARCH-R1-S1
SET P027 P006
SSFTON P027
SMOVL C00164 BC00164 V=100.0  +MOVJ EC00164
SREFP 3 C00165 BC00165  +REFP EC00165
CALL JOB:SEARCH-R1-S1
SET P027 P006
SSFTON P027
SMOVL C00166 BC00166 V=133.3  +MOVJ EC00166
SSFTOF
SMOVL C00167 BC00167 V=266.7  +MOVJ EC00167
SMOVL C00168 BC00168 V=100.0  +MOVJ EC00168
SREFP 3 C00169 BC00169  +REFP EC00169
CALL JOB:SEARCH-R1-S1
SET P028 P006
SSFTON P028
SMOVL C00170 BC00170 V=100.0  +MOVJ EC00170
SREFP 3 C00171 BC00171  +REFP EC00171
CALL JOB:SEARCH-R1-S1
SET P028 P006
SSFTON P028
SMOVL C00172 BC00172 V=133.3  +MOVJ EC00172
SSFTOF
PAUSE
MACRO1 MJ#(0) ARGF14
SSFTON P028
SMOVL C00173 BC00173 V=100.0  +MOVJ EC00173
ARCON
SWVON WEV#(50)
SSFTON P027
SMOVL C00174 BC00174 V=9.2  +MOVJ EC00174
ARCOF
SWVOF
SMOVL C00175 BC00175 V=100.0  +MOVJ EC00175
SSFTOF
SMOVL C00176 BC00176 V=100.0  +MOVJ EC00176
MACRO1 MJ#(0) ARGF6
SMOVL C00177 BC00177 V=266.7  +MOVJ EC00177
SSFTON P025
SMOVL C00178 BC00178 V=100.0  +MOVJ EC00178
ARCON
SWVON WEV#(50)
SSFTON P026
SMOVL C00179 BC00179 V=6.7  +MOVJ EC00179
SMOVL C00180 BC00180 V=6.7  +MOVJ EC00180
ARCOF
SWVOF
SMOVL C00181 BC00181 V=133.3  +MOVJ EC00181
SSFTOF
SMOVL C00182 BC00182 V=666.7  +MOVJ EC00182
MOVJ C00183 BC00183 VJ=100.00  +MOVJ EC00183 VJ=100.00
MOVJ C00184 BC00184 VJ=100.00  +MOVJ EC00184 VJ=100.00
MOVJ C00185 BC00185 VJ=100.00  +MOVJ EC00185 VJ=100.00
MOVJ C00186 BC00186 VJ=100.00  +MOVJ EC00186 VJ=100.00
SMOVL C00187 BC00187 V=333.3  +MOVJ EC00187
SSFTON P031
SMOVL C00188 BC00188 V=100.0  +MOVJ EC00188
ARCON
SSFTON P032
SMOVL C00189 BC00189 V=11.0  +MOVJ EC00189
ARCOF
SMOVL C00190 BC00190 V=266.7  +MOVJ EC00190
SSFTOF
SMOVL C00191 BC00191 V=266.7  +MOVJ EC00191
SSFTON P033
SMOVL C00192 BC00192 V=100.0  +MOVJ EC00192
ARCON
SMOVL C00193 BC00193 V=11.0  +MOVJ EC00193
SSFTON P024
SMOVL C00194 BC00194 V=11.0  +MOVJ EC00194
SMOVL C00195 BC00195 V=11.0  +MOVJ EC00195
ARCOF
SMOVL C00196 BC00196 V=266.7  +MOVJ EC00196
SSFTOF
SMOVL C00197 BC00197 V=266.7  +MOVJ EC00197
SMOVL C00198 BC00198 V=266.7  +MOVJ EC00198
MOVJ C00199 BC00199 VJ=100.00  +MOVJ EC00199 VJ=100.00
END
